Yaskawa INFORM job: sDrill44_(14).JBI

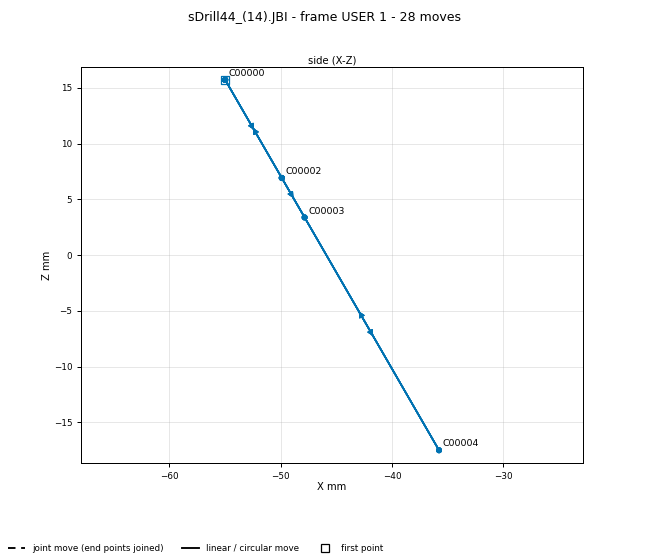
[picture p0: tool path of sDrill44_(14).JBI in frame USER 1, 28 of 28 moves have a stored position in this frame; points joined in program order, loops and branches not executed]
/JOB
//NAME sDrill44_(14)
//POS
///NPOS 7,0,0,0,0,0
///USER 1
///TOOL 3
///POSTYPE USER
///RECTAN
///RCONF 1,0,0,0,0,0
C00000=1.964,-29.946,15.742,-90.000,-150.794,-116.565
C00001=1.964,-29.946,15.742,-90.000,-150.794,-116.565
C00002=1.964,-24.866,6.943,-90.000,-150.794,-116.565
C00003=1.964,-22.817,3.394,-90.000,-150.794,-116.565
C00004=1.964,-11.000,-17.074,-90.000,-150.794,-116.565
C00005=1.964,-24.866,6.943,-90.000,-150.794,-116.565
C00006=1.964,-29.946,15.742,-90.000,-150.794,-116.565
C00000=54.944,0.008,15.743,0.000,-152.507,-33.690
C00001=54.944,0.008,15.743,0.000,-152.507,-33.690
C00002=49.864,0.008,6.944,0.000,-152.507,-33.690
C00003=47.815,0.008,3.395,0.000,-152.507,-33.690
C00004=35.788,0.008,-17.436,0.000,-152.507,-33.690
C00005=49.864,0.008,6.944,0.000,-152.507,-33.690
C00006=54.944,0.008,15.743,0.000,-152.507,-33.690
C00000=-0.401,29.967,15.730,90.000,-150.794,63.435
C00001=-0.401,29.967,15.730,90.000,-150.794,63.435
C00002=-0.401,24.887,6.931,90.000,-150.794,63.435
C00003=-0.401,22.838,3.382,90.000,-150.794,63.435
C00004=-0.401,10.773,-17.515,90.000,-150.794,63.435
C00005=-0.401,24.887,6.931,90.000,-150.794,63.435
C00006=-0.401,29.967,15.730,90.000,-150.794,63.435
C00000=-54.968,2.694,15.730,180.000,-152.507,146.310
C00001=-54.968,2.694,15.730,180.000,-152.507,146.310
C00002=-49.888,2.694,6.931,180.000,-152.507,146.310
C00003=-47.838,2.694,3.382,180.000,-152.507,146.310
C00004=-35.773,2.694,-17.515,180.000,-152.507,146.310
C00005=-49.888,2.694,6.931,180.000,-152.507,146.310
C00006=-54.968,2.694,15.730,180.000,-152.507,146.310
//INST
///ATTR SC,RW,RJ
////FRAME USER 1
///GROUP1 RB1
///LVARS 2,0,0,0,0,0,0,0
NOP
SET LB000 1
SET LB001 25
MOVJ C00000 VJ=17
' Cutting Move Starts
MOVL C00001 V=17 PL=LB000 ACC=LB001 DEC=LB001
MOVL C00002 V=17 PL=LB000 ACC=LB001 DEC=LB001
MOVL C00003 V=17 PL=LB000 ACC=LB001 DEC=LB001
MOVL C00004 V=7 PL=LB000 ACC=LB001 DEC=LB001
MOVL C00005 V=17 PL=LB000 ACC=LB001 DEC=LB001
' Rapid Move Starts
MOVL C00006 V=17 PL=LB000 ACC=LB001 DEC=LB001
' By Autodesk Fusion CAM 2.0.20494
' Tool = 3
' Spindle = 5000 RPM
' Set Position Level
' Set Acceleration
' Program Start
' First Toolpath Point
' Last Toolpath Point
MOVJ C00000 VJ=17
' Cutting Move Starts
MOVL C00001 V=17 PL=LB000 ACC=LB001 DEC=LB001
MOVL C00002 V=17 PL=LB000 ACC=LB001 DEC=LB001
MOVL C00003 V=17 PL=LB000 ACC=LB001 DEC=LB001
MOVL C00004 V=7 PL=LB000 ACC=LB001 DEC=LB001
MOVL C00005 V=17 PL=LB000 ACC=LB001 DEC=LB001
' Rapid Move Starts
MOVL C00006 V=17 PL=LB000 ACC=LB001 DEC=LB001
' By Autodesk Fusion CAM 2.0.20494
' Tool = 3
' Spindle = 5000 RPM
' Set Position Level
' Set Acceleration
' Program Start
' First Toolpath Point
' Last Toolpath Point
MOVJ C00000 VJ=17
' Cutting Move Starts
MOVL C00001 V=17 PL=LB000 ACC=LB001 DEC=LB001
MOVL C00002 V=17 PL=LB000 ACC=LB001 DEC=LB001
MOVL C00003 V=17 PL=LB000 ACC=LB001 DEC=LB001
MOVL C00004 V=7 PL=LB000 ACC=LB001 DEC=LB001
MOVL C00005 V=17 PL=LB000 ACC=LB001 DEC=LB001
' Rapid Move Starts
MOVL C00006 V=17 PL=LB000 ACC=LB001 DEC=LB001
' By Autodesk Fusion CAM 2.0.20494
' Tool = 3
' Spindle = 5000 RPM
' Set Position Level
' Set Acceleration
' Program Start
' First Toolpath Point
' Last Toolpath Point
MOVJ C00000 VJ=17
' Cutting Move Starts
MOVL C00001 V=17 PL=LB000 ACC=LB001 DEC=LB001
MOVL C00002 V=17 PL=LB000 ACC=LB001 DEC=LB001
MOVL C00003 V=17 PL=LB000 ACC=LB001 DEC=LB001
MOVL C00004 V=7 PL=LB000 ACC=LB001 DEC=LB001
MOVL C00005 V=17 PL=LB000 ACC=LB001 DEC=LB001
' Rapid Move Starts
MOVL C00006 V=17 PL=LB000 ACC=LB001 DEC=LB001
' By Autodesk Fusion CAM 2.0.20494
' Tool = 3
' Spindle = 5000 RPM
' Set Position Level
' Set Acceleration
' Program Start
' First Toolpath Point
END
